Staubli VAL3: sRobot2fRobot.pgx

program sRobot2fRobot()
begin

  //没有ClearBuffer 这个比较难联通
  clearBuffer(sClient)

  //把客户端收到不为空的信息通过服务器传送出去
  while true
    //服务器
    //clearBuffer(sServer)

    call ClientGet(sSecondRStatus)
    //popUpMsg(sFirstRStatus)

    delay(0)
  endWhile

end
